(* PLC project FirstProject, ps_m.k. Beremiz 1 *)
(* stored: creationDateTime 2019-10-22T21:12:26, modificationDateTime 2019-11-28T01:52:46 *)

FUNCTION_BLOCK C_Pragma
  VAR_INPUT
    OUT : INT := 25;
  END_VAR
  VAR_OUTPUT
    VALUE : INT := 0;
  END_VAR
  VAR_INPUT
    IN : INT := 24;
    PERMIT : INT := 1;
  END_VAR

            {{
    extern void WritePin(int, int);
    extern void InitPin(int, int);
    extern void CheckPin();
    extern int ReadPin(int);
    
    CheckPin();
    InitPin(24, 0);
    InitPin(25, 1);
    if (GetFbVar(PERMIT) > 0) {
      WritePin(25, ReadPin(24));
    }
}}
          
END_FUNCTION_BLOCK

PROGRAM plc_prg
  VAR_INPUT
    Input : INT := 24;
    Output : INT := 25;
  END_VAR
  VAR
    C_Pragma0 : C_Pragma;
  END_VAR

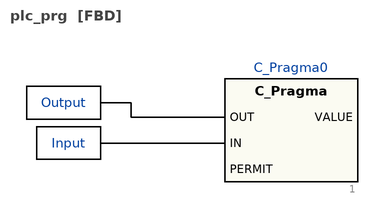
(* FBD diagram, written out as Structured Text *)
C_Pragma0(OUT := Output, IN := Input);
END_PROGRAM

CONFIGURATION config
  RESOURCE resource1 ON PLC
    TASK GetTimeSync(INTERVAL := T#0.15ms, PRIORITY := 0);
    PROGRAM plc_task_instance WITH GetTimeSync : plc_prg;
  END_RESOURCE
END_CONFIGURATION
